TYPE ST_CircuitBreakerHMI :
STRUCT
    stCommand: ST_CircuitBreakerCommand;        // Komutlar
    stStatus: ST_CircuitBreakerStatus;          // Durum bilgileri
    stConfig: ST_CircuitBreakerConfig;          // Konfigürasyon
    stStatistics: ST_CircuitBreakerStatistics;  // İstatistik verileri
END_STRUCT
END_TYPE

(* stored: Version 1.1.0.1, ProductVersion 3.1.4024.15
   DUT ST_CircuitBreakerHMI: Id {e0701674-969d-4c24-b614-9a74dd78f07d} *)
